FUNCTION_BLOCK Rec_Queue
VAR_INPUT
END_VAR
VAR_IN_OUT
	REC_Queue_List     : ARRAY[0..Param_Queue.MAX_QUEUE_SIZE] OF REC_CMD_DATA;
END_VAR
VAR_OUTPUT
	Err_Out            : BOOL;
END_VAR
VAR
	Head_Var           : INT;
	Tail_Var           : INT;
	Count_Var          : INT;
	Index_Init         : INT;
	Del_QueueTemp      : REC_CMD_DATA;
	Init_QueueTemp     : REC_CMD_DATA;
END_VAR

METHOD PUBLIC Count_Queue : INT;
VAR_INPUT
END_VAR
Count_Queue := Count_Var;
END_METHOD

METHOD PUBLIC Delete_Queue : REC_CMD_DATA;
VAR_INPUT
END_VAR
IF Count_Var = 0 THEN
	Err_Out:= TRUE;
	RETURN;
ELSE
	Err_Out:= FALSE;
	Count_Var:= Count_Var-1; 
	Del_QueueTemp:= REC_Queue_List[Head_Var];
	Head_Var:= (Head_Var +1) MOD Param_Queue.MAX_QUEUE_SIZE;
	Delete_Queue:= Del_QueueTemp;
END_IF
END_METHOD

METHOD PUBLIC Empty_Queue : BOOL;
VAR_INPUT
END_VAR
IF Count_Var = 0 THEN
	Empty_Queue:= TRUE;
ELSE 
	Empty_Queue:= FALSE;
END_IF
END_METHOD

METHOD PUBLIC Full_Queue: BOOL;
VAR_INPUT
END_VAR
IF Count_Var = Param_Queue.MAX_QUEUE_SIZE THEN
	Full_Queue := TRUE;
ELSE
	Full_Queue := FALSE;
END_IF
END_METHOD

METHOD PUBLIC Head_Queue : REC_CMD_DATA;
VAR_INPUT
END_VAR
Head_Queue:= REC_Queue_List[Head_Var];
END_METHOD

METHOD PUBLIC Init_Queue
VAR_INPUT
END_VAR
Head_Var:= 0;
Tail_Var:= 0;
Count_Var:= 0;
Err_Out:= FALSE;
Del_QueueTemp:= Init_QueueTemp;
FOR Index_Init:=0 TO Param_Queue.MAX_QUEUE_SIZE BY 1 DO
	REC_Queue_List[Index_Init]:= Init_QueueTemp;
END_FOR
END_METHOD

METHOD PUBLIC Insert_Queue
VAR_INPUT
	Insert_Queue : REC_CMD_DATA;
END_VAR
IF Count_Var= Param_Queue.MAX_QUEUE_SIZE THEN
	Err_Out:= TRUE;
	RETURN;
ELSE
	Err_Out:= FALSE;
	Count_Var:= Count_Var + 1;
	REC_Queue_List[Tail_Var]:= Insert_Queue;
	Tail_Var:= (Tail_Var +1) MOD Param_Queue.MAX_QUEUE_SIZE;
END_IF
END_METHOD

END_FUNCTION_BLOCK

(* stored: Version 1.1.0.1, ProductVersion 3.1.4018.5
   POU Rec_Queue: Id {918628db-52ec-4ebd-a8e0-f75cd21824a9}, SpecialFunc None
   Method Count_Queue: Id {e0d8f68d-9c9f-4d00-aff9-42432decdadc}
   Method Delete_Queue: Id {01156375-bf24-4bcd-8356-890c29f166df}
   Method Empty_Queue: Id {254d9fc6-b70b-45b7-957a-e33af6ccc0ee}
   Method Full_Queue: Id {52406aae-b632-45e9-85fd-469246537349}
   Method Head_Queue: Id {0d502f0c-ca5c-4ef3-8605-074a52a1e085}
   Method Init_Queue: Id {9a8d14a0-daef-4c7e-ac44-14fe5b7653ba}
   Method Insert_Queue: Id {da424955-1440-4185-8547-de1608264453} *)
